Staubli VAL3: BuildTitle.pgx

program BuildTitle(string x_sTitle, string x_sOptional)
  local string l_sTitle
begin
  // This program add the conveyor calibration file name
  // to the title
  call up:strAlign(x_sOptional,8,"R","═")
  call up:strAlign(x_sTitle,29,"L","═")
  l_sTitle=x_sTitle+x_sOptional
  title(l_sTitle)
end
